"Z2RFRO1"	Q 38.0	BOOL	// [Z2ZB.M07]: SAFETY COMMON 1 (RESERVA)
"Z2RFRO2"	Q 38.1	BOOL	// [Z2ZB.M07]: SAFETY COMMON 2 (Z2ES)
"Z2ZB_M07_R1"	Q 38.2	BOOL	// [Z2ZB.M07]: RESERVA
"Z2EV7b"	Q 38.3	BOOL	// [Z2ZB.M07]: Z2 EV 7 bar
"Z3RFRO1"	Q 47.0	BOOL	// (Z2ZB.M09): RELE COMUN DE SEGURIDAD (Z3AU)
"Z3RFRO2"	Q 47.1	BOOL	// (Z2ZB.M09): RELE COMUN DE SEGURIDAD (Z3ES)
"Z3EV7B"	Q 47.3	BOOL	// (Z2ZB.M09): EV 7 BARS
"A0SB_M04_R1"	Q 70.0	BOOL	// [A0SB.M04]: RESERVA
"A0SB_M04_R2"	Q 70.1	BOOL	// [A0SB.M04]: RESERVA
"A0SB_M04_R3"	Q 70.2	BOOL	// [A0SB.M04]: RESERVA
"A0SB_M04_R4"	Q 70.3	BOOL	// [A0SB.M04]: RESERVA
"A0SB_M04_R5"	Q 70.4	BOOL	// [A0SB.M04]: RESERVA
"A0SB_M04_R6"	Q 70.5	BOOL	// [A0SB.M04]: RESERVA
"A0SB_M04_R7"	Q 70.6	BOOL	// [A0SB.M04]: RESERVA
"A0SB_M04_R8"	Q 70.7	BOOL	// [A0SB.M04]: RESERVA
"A0VAT"	Q 71.0	BOOL	// [A0SB.M06]: A0 WORK AUTHORIZATION LAMP 1 (GREEN)
"A0VIT"	Q 71.1	BOOL	// [A0SB.M06]: A0 WORK PROHIBITION LAMP 1 (RED)
"A0VDF"	Q 71.2	BOOL	// [A0SB.M06]: A0 DEFAULT LAMP 1 (ORANGE)
"A0SB_M06_R1"	Q 71.3	BOOL	// [A0SB.M06]: RESERVA
"A0SB_M06_R2"	Q 71.4	BOOL	// [A0SB.M06]: RESERVA
"A0SB_M06_R3"	Q 71.5	BOOL	// [A0SB.M06]: RESERVA
"A0SB_M06_R4"	Q 71.6	BOOL	// [A0SB.M06]: RESERVA
"A0SB_M06_R5"	Q 71.7	BOOL	// [A0SB.M06]: RESERVA
"A0RFRO1"	Q 90.0	BOOL	// [A0SB.M11]: A0 SAFETY COMMON 3 (FRO1)
"A0RFRO2"	Q 90.1	BOOL	// [A0SB.M11]: A0 SAFETY COMMON 4 (FRO2)
"A0RFRO3"	Q 90.2	BOOL	// [A0SB.M11]: A0 SAFETY COMMON 5 (FRO3)
"A0SB_M11_R1"	Q 90.3	BOOL	// [A0SB.M11]: RESERVA
"B0SB_M04_R1"	Q 110.0	BOOL	// [B0SB.M04]: RESERVA
"B0SB_M04_R2"	Q 110.1	BOOL	// [B0SB.M04]: RESERVA
"B0SB_M04_R3"	Q 110.2	BOOL	// [B0SB.M04]: RESERVA
"B0SB_M04_R4"	Q 110.3	BOOL	// [B0SB.M04]: RESERVA
"B0SB_M04_R5"	Q 110.4	BOOL	// [B0SB.M04]: RESERVA
"B0SB_M04_R6"	Q 110.5	BOOL	// [B0SB.M04]: RESERVA
"B0SB_M04_R7"	Q 110.6	BOOL	// [B0SB.M04]: RESERVA
"B0SB_M04_R8"	Q 110.7	BOOL	// [B0SB.M04]: RESERVA
"B0VAT"	Q 111.0	BOOL	// [B0SB.M06]: B0 WORK AUTHORIZATION LAMP 1 (GREEN)
"B0VIT"	Q 111.1	BOOL	// [B0SB.M06]: B0 WORK PROHIBITION LAMP 1 (RED)
"B0VDF"	Q 111.2	BOOL	// [B0SB.M06]: B0 DEFAULT LAMP 1 (ORANGE)
"B0SB_M06_R1"	Q 111.3	BOOL	// [B0SB.M06]: RESERVA
"B0SB_M06_R2"	Q 111.4	BOOL	// [B0SB.M06]: RESERVA
"B0SB_M06_R3"	Q 111.5	BOOL	// [B0SB.M06]: RESERVA
"B0SB_M06_R4"	Q 111.6	BOOL	// [B0SB.M06]: RESERVA
"B0SB_M06_R5"	Q 111.7	BOOL	// [B0SB.M06]: RESERVA
"B0SB_M11_R1"	Q 130.3	BOOL	// [B0SB.M11]: RESERVA
"C0SB_M04_R1"	Q 150.0	BOOL	// [C0SB.M04]: RESERVA
"C0SB_M04_R2"	Q 150.1	BOOL	// [C0SB.M04]: RESERVA
"C0SB_M04_R3"	Q 150.2	BOOL	// [C0SB.M04]: RESERVA
"C0SB_M04_R4"	Q 150.3	BOOL	// [C0SB.M04]: RESERVA
"C0SB_M04_R5"	Q 150.4	BOOL	// [C0SB.M04]: RESERVA
"C0SB_M04_R6"	Q 150.5	BOOL	// [C0SB.M04]: RESERVA
"C0SB_M04_R7"	Q 150.6	BOOL	// [C0SB.M04]: RESERVA
"C0SB_M04_R8"	Q 150.7	BOOL	// [C0SB.M04]: RESERVA
"C0VAT"	Q 151.0	BOOL	// [C0SB.M06]: C0 WORK AUTHORIZATION LAMP 1 (GREEN)
"C0VIT"	Q 151.1	BOOL	// [C0SB.M06]: C0 WORK PROHIBITION LAMP 1 (RED)
"C0VDF"	Q 151.2	BOOL	// [C0SB.M06]: C0 DEFAULT LAMP 1 (ORANGE)
"C0SB_M06_R1"	Q 151.3	BOOL	// [C0SB.M06]: RESERVA
"C0SB_M06_R2"	Q 151.4	BOOL	// [C0SB.M06]: RESERVA
"C0SB_M06_R3"	Q 151.5	BOOL	// [C0SB.M06]: RESERVA
"C0SB_M06_R4"	Q 151.6	BOOL	// [C0SB.M06]: RESERVA
"C0SB_M06_R5"	Q 151.7	BOOL	// [C0SB.M06]: RESERVA
"C0SB_M11_R1"	Q 170.3	BOOL	// [C0SB.M11]: RESERVA
"D0SB_M04_R1"	Q 190.0	BOOL	// [D0SB.M04]: RESERVA
"D0SB_M04_R2"	Q 190.1	BOOL	// [D0SB.M04]: RESERVA
"D0SB_M04_R3"	Q 190.2	BOOL	// [D0SB.M04]: RESERVA
"D0SB_M04_R4"	Q 190.3	BOOL	// [D0SB.M04]: RESERVA
"D0SB_M04_R5"	Q 190.4	BOOL	// [D0SB.M04]: RESERVA
"D0SB_M04_R6"	Q 190.5	BOOL	// [D0SB.M04]: RESERVA
"D0SB_M04_R7"	Q 190.6	BOOL	// [D0SB.M04]: RESERVA
"D0SB_M04_R8"	Q 190.7	BOOL	// [D0SB.M04]: RESERVA
"D0VAT"	Q 191.0	BOOL	// [D0SB.M06]: D0 WORK AUTHORIZATION LAMP 1 (GREEN)
"D0VIT"	Q 191.1	BOOL	// [D0SB.M06]: D0 WORK PROHIBITION LAMP 1 (RED)
"D0VDF"	Q 191.2	BOOL	// [D0SB.M06]: D0 DEFAULT LAMP 1 (ORANGE)
"D0LPDPY"	Q 191.3	BOOL	// [D0SB.M06]: LAMPADA DEFEITO POKAYOKE
"D0SRDPY"	Q 191.4	BOOL	// [D0SB.M06]: SIRENE DEFEITO POKAYOKE
"TR0VAT"	Q 191.5	BOOL	// [D0SB.M06]: TR0 LAMP(GREEN)
"TR0VIT"	Q 191.6	BOOL	// [D0SB.M06]: TR0 LAMP (RED)
"D0SB_M06_R5"	Q 191.7	BOOL	// [D0SB.M06]: RESERVA
"D0RFRO1"	Q 210.0	BOOL	// [D0SB.M11]: D0 SAFETY COMMON 3 (FRO1)
"D0RFRO2"	Q 210.1	BOOL	// [D0SB.M11]: D0 SAFETY COMMON 4 (FRO2)
"D0RFRO3"	Q 210.2	BOOL	// [D0SB.M11]: D0 SAFETY COMMON 5 (FRO3)
"D0SB_M11_R1"	Q 210.3	BOOL	// [D0SB.M11]: RESERVA
"E0SB_M04_R1"	Q 230.0	BOOL	// [E0SB.M04]: RESERVA
"E0SB_M04_R2"	Q 230.1	BOOL	// [E0SB.M04]: RESERVA
"E0SB_M04_R3"	Q 230.2	BOOL	// [E0SB.M04]: RESERVA
"E0SB_M04_R4"	Q 230.3	BOOL	// [E0SB.M04]: RESERVA
"E0SB_M04_R5"	Q 230.4	BOOL	// [E0SB.M04]: RESERVA
"E0SB_M04_R6"	Q 230.5	BOOL	// [E0SB.M04]: RESERVA
"E0SB_M04_R7"	Q 230.6	BOOL	// [E0SB.M04]: RESERVA
"E0SB_M04_R8"	Q 230.7	BOOL	// [E0SB.M04]: RESERVA
"E0VAT"	Q 231.0	BOOL	// [E0SB.M06]: E0 WORK AUTHORIZATION LAMP 1 (GREEN)
"E0VIT"	Q 231.1	BOOL	// [E0SB.M06]: E0 WORK PROHIBITION LAMP 1 (RED)
"E0VDF"	Q 231.2	BOOL	// [E0SB.M06]: E0 DEFAULT LAMP 1 (ORANGE)
"E0SB_M06_R1"	Q 231.3	BOOL	// [E0SB.M06]: RESERVA
"E0SB_M06_R2"	Q 231.4	BOOL	// [E0SB.M06]: RESERVA
"E0SB_M06_R3"	Q 231.5	BOOL	// [E0SB.M06]: RESERVA
"E0SB_M06_R4"	Q 231.6	BOOL	// [E0SB.M06]: RESERVA
"E0SB_M06_R5"	Q 231.7	BOOL	// [E0SB.M06]: RESERVA
"E0SB_M11_R1"	Q 250.3	BOOL	// [E0SB.M11]: RESERVA
"F0SB_M04_R1"	Q 270.0	BOOL	// [F0SB.M04]: RESERVA
"F0SB_M04_R2"	Q 270.1	BOOL	// [F0SB.M04]: RESERVA
"F0SB_M04_R3"	Q 270.2	BOOL	// [F0SB.M04]: RESERVA
"F0SB_M04_R4"	Q 270.3	BOOL	// [F0SB.M04]: RESERVA
"F0SB_M04_R5"	Q 270.4	BOOL	// [F0SB.M04]: RESERVA
"F0SB_M04_R6"	Q 270.5	BOOL	// [F0SB.M04]: RESERVA
"F0SB_M04_R7"	Q 270.6	BOOL	// [F0SB.M04]: RESERVA
"F0SB_M04_R8"	Q 270.7	BOOL	// [F0SB.M04]: RESERVA
"F0VAT"	Q 271.0	BOOL	// [F0SB.M06]: F0 WORK AUTHORIZATION LAMP 1 (GREEN)
"F0VIT"	Q 271.1	BOOL	// [F0SB.M06]: F0 WORK PROHIBITION LAMP 1 (RED)
"F0VDF"	Q 271.2	BOOL	// [F0SB.M06]: F0 DEFAULT LAMP 1 (ORANGE)
"F0SB_M06_R1"	Q 271.3	BOOL	// [F0SB.M06]: RESERVA
"F0SB_M06_R2"	Q 271.4	BOOL	// [F0SB.M06]: RESERVA
"F0SB_M06_R3"	Q 271.5	BOOL	// [F0SB.M06]: RESERVA
"F0SB_M06_R4"	Q 271.6	BOOL	// [F0SB.M06]: RESERVA
"F0SB_M06_R5"	Q 271.7	BOOL	// [F0SB.M06]: RESERVA
"F0RFRO1"	Q 290.0	BOOL	// [F0SB.M11]: F0 SAFETY COMMON 3 (F0SOP)
"F0RFRO2"	Q 290.1	BOOL	// [F0SB.M11]: F0 SAFETY COMMON 4 (F0)
"F0RFRO3"	Q 290.2	BOOL	// [F0SB.M11]: F0 SAFETY COMMON 5 (F0)
"F0SB_M11_R1"	Q 290.3	BOOL	// [F0SB.M11]: RESERVA
"G0SB_M04_R1"	Q 310.0	BOOL	// [G0SB.M04]: RESERVA
"G0SB_M04_R2"	Q 310.1	BOOL	// [G0SB.M04]: RESERVA
"G0SB_M04_R3"	Q 310.2	BOOL	// [G0SB.M04]: RESERVA
"G0SB_M04_R4"	Q 310.3	BOOL	// [G0SB.M04]: RESERVA
"G0SB_M04_R5"	Q 310.4	BOOL	// [G0SB.M04]: RESERVA
"G0SB_M04_R6"	Q 310.5	BOOL	// [G0SB.M04]: RESERVA
"G0SB_M04_R7"	Q 310.6	BOOL	// [G0SB.M04]: RESERVA
"G0SB_M04_R8"	Q 310.7	BOOL	// [G0SB.M04]: RESERVA
"G0VAT"	Q 311.0	BOOL	// [G0SB.M06]: G0 WORK AUTHORIZATION LAMP 1 (GREEN)
"G0VIT"	Q 311.1	BOOL	// [G0SB.M06]: G0 WORK PROHIBITION LAMP 1 (RED)
"G0VDF"	Q 311.2	BOOL	// [G0SB.M06]: G0 DEFAULT LAMP 1 (ORANGE)
"G0SB_M06_R1"	Q 311.3	BOOL	// [G0SB.M06]: RESERVA
"G0SB_M06_R2"	Q 311.4	BOOL	// [G0SB.M06]: RESERVA
"G0SB_M06_R3"	Q 311.5	BOOL	// [G0SB.M06]: RESERVA
"G0SB_M06_R4"	Q 311.6	BOOL	// [G0SB.M06]: RESERVA
"G0SB_M06_R5"	Q 311.7	BOOL	// [G0SB.M06]: RESERVA
"G0SB_M11_R1"	Q 330.3	BOOL	// [G0SB.M11]: RESERVA
"K0SB_M04_R1"	Q 380.0	BOOL	// [K0SB.M04]: RESERVA
"K0SB_M04_R2"	Q 380.1	BOOL	// [K0SB.M04]: RESERVA
"K0SB_M04_R3"	Q 380.2	BOOL	// [K0SB.M04]: RESERVA
"K0SB_M04_R4"	Q 380.3	BOOL	// [K0SB.M04]: RESERVA
"K0SB_M04_R5"	Q 380.4	BOOL	// [K0SB.M04]: RESERVA
"K0SB_M04_R6"	Q 380.5	BOOL	// [K0SB.M04]: RESERVA
"K0SB_M04_R7"	Q 380.6	BOOL	// [K0SB.M04]: RESERVA
"KOSB_M04_R8"	Q 380.7	BOOL	// [K0SB.M04]: RESERVA
"K0VAT"	Q 381.0	BOOL	// [K0SB.M06]: C0 WORK AUTHORIZATION LAMP 1 (GREEN)
"K0VIT"	Q 381.1	BOOL	// [K0SB.M06]: C0 WORK PROHIBITION LAMP 1 (RED)
"K0VDF"	Q 381.2	BOOL	// [K0SB.M06]: C0 DEFAULT LAMP 1 (ORANGE)
"K0SB_M06_R1"	Q 381.3	BOOL	// [K0SB.M06]: RESERVA
"K0SB_M06_R2"	Q 381.4	BOOL	// [K0SB.M06]: RESERVA
"K0SB_M06_R3"	Q 381.5	BOOL	// [K0SB.M06]: RESERVA
"K0SB_M06_R4"	Q 381.6	BOOL	// [K0SB.M06]: RESERVA
"K0SB_M06_R5"	Q 381.7	BOOL	// [K0SB.M06]: RESERVA
"K0RFRO1"	Q 400.0	BOOL	// [K0SB.M11]: K0 SAFETY COMMON 3 (K0SOP)
"K0RFRO2"	Q 400.1	BOOL	// [K0SB.M11]: K0 SAFETY COMMON 4 (K0SOP)
"K0RFRO3"	Q 400.2	BOOL	// [K0SB.M11]: K0 SAFETY COMMON 5 (K0SOP)
"K0SB_M11_R1"	Q 400.3	BOOL	// [K0SB.M11]: RESERVA
"A0EAPLA"	Q 500.0	BOOL	// [A0IM1.A0S11]: A0: EV AVANÇO PILOTO A
"A0EASRB"	Q 500.1	BOOL	// [A0IM1.A0S11]: A0: EV AVANÇO SERRAGE MANUAL B
"A0IM_A0S11_R1"	Q 500.2	BOOL	// [A0IM1.A0S11]: RESERVA
"A0EASRD"	Q 500.3	BOOL	// [A0IM1.A0S11]: A0: EV AVANÇO SERRAGE D
"A0ERPLA"	Q 500.4	BOOL	// [A0IM1.A0S11]: A0: EV RECUO PILOTO A
"A0ERSRB"	Q 500.5	BOOL	// [A0IM1.A0S11]: A0: EV RECUO SERRAGE MANUAL B
"A0IM_A0S11_R2"	Q 500.6	BOOL	// [A0IM1.A0S11]: RESERVA
"A0ERSRD"	Q 500.7	BOOL	// [A0IM1.A0S11]: A0: EV RECUO SERRAGE D
"A0EAPLE"	Q 501.0	BOOL	// [A0IM1.A0S12]: A0: EV AVANÇO PILOTO E
"A0IM_A0S12_R5"	Q 501.1	BOOL	// [A0IM1.A0S12]: RESERVA
"A0IM_A0S12_R3"	Q 501.2	BOOL	// [A0IM1.A0S12]: RESERVA
"A0IM_A0S12_R4"	Q 501.3	BOOL	// [A0IM1.A0S12]: RESERVA
"A0ERPLE"	Q 501.4	BOOL	// [A0IM1.A0S12]: A0: EV RECUO PILOTO E
"A0IM_A0S12_R6"	Q 501.5	BOOL	// [A0IM1.A0S12]: RESERVA
"A0IM_A0S12_R7"	Q 501.6	BOOL	// [A0IM1.A0S12]: RESERVA
"A0IM_A0S12_R8"	Q 501.7	BOOL	// [A0IM1.A0S12]: RESERVA
"B0EAPLA"	Q 520.0	BOOL	// [B0IM1.B0S11]: B0: EV AVANÇO PILOTO A
"B0EASRB"	Q 520.1	BOOL	// [B0IM1.B0S11]: B0: EV AVANÇO SERRAGE B
"B0IM_B0S11_R1"	Q 520.2	BOOL	// [B0IM1.B0S11]: RESERVA
"B0IM_B0S11_R2"	Q 520.3	BOOL	// [B0IM1.B0S11]: RESERVA
"B0ERPLA"	Q 520.4	BOOL	// [B0IM1.B0S11]: B0: EV RECUO PILOTO A
"B0ERSRB"	Q 520.5	BOOL	// [B0IM1.B0S11]: D0: EV RECUO SERRAGE B
"B0IM_B0S11_R3"	Q 520.6	BOOL	// [B0IM1.B0S11]: RESERVA
"B0IM_B0S11_R4"	Q 520.7	BOOL	// [B0IM1.B0S11]: RESERVA
"D0EAPLA"	Q 560.0	BOOL	// [D0IM1.D0S11]: D0: EV AVANÇO PILOTO A
"D0EACAB"	Q 560.1	BOOL	// [D0IM1.D0S11]: D0:EV AVANÇO CARRO B
"D0EASRC"	Q 560.2	BOOL	// [D0IM1.D0S11]: D0: EV AVANÇO SERRAGE C
"D0EASRD"	Q 560.3	BOOL	// [D0IM1.D0S11]: D0: EV AVANÇO SERRAGE D
"D0ERPLA"	Q 560.4	BOOL	// [D0IM1.D0S11]: D0: EV RECUO PILOTO A
"D0ERCAB"	Q 560.5	BOOL	// [D0IM1.D0S11]: D0:EV RECUO CARRO B
"D0ERSRC"	Q 560.6	BOOL	// [D0IM1.D0S11]: D0: EV RECUO SERRAGE C
"D0ERSRD"	Q 560.7	BOOL	// [D0IM1.D0S11]: D0: EV RECUO SERRAGE D
"D0EACAB1"	Q 561.0	BOOL	// [D0IM1.D0S12]: D0:EV FREIO D0CAB1
"D0EAPLE"	Q 561.1	BOOL	// [D0IM1.D0S12]: D0: EV AVANÇO PILOTO E
"D0EASRMF"	Q 561.2	BOOL	// [D0IM1.D0S12]:  ElectroValvula Avance SRM1
"D0IM_D0S12_R4"	Q 561.3	BOOL	// [D0IM1.D0S12]: RESERVA
"D0ERCAB1"	Q 561.4	BOOL	// [D0IM1.D0S12]: D0:EV RECUO CARRO B1 (FREIO)
"D0ERPLE"	Q 561.5	BOOL	// [D0IM1.D0S12]: D0: EV RECUO PILOTO E
"D0ERSRMF"	Q 561.6	BOOL	// [D0IM1.D0S12]: [D0IM1.D0S12]:  ElectroValvula Retroceso SRM1
"D0IM_D0S12_R8"	Q 561.7	BOOL	// [D0IM1.D0S12]: RESERVA
"E0EAPLA"	Q 580.0	BOOL	// [E0IM1.E0S11]: E0: EV AVANÇO PILOTO A
"E0EASRB"	Q 580.1	BOOL	// [E0IM1.E0S11]: E0: EV AVANÇO SERRAGE B
"E0IM_E0S11_R1"	Q 580.2	BOOL	// [E0IM1.E0S11]: RESERVA
"E0IM_E0S11_R2"	Q 580.3	BOOL	// [E0IM1.E0S11]: RESERVA
"E0ERPLA"	Q 580.4	BOOL	// [E0IM1.E0S11]: E0: EV RECUO PILOTO A
"E0ERSRB"	Q 580.5	BOOL	// [E0IM1.E0S11]: E0: EV RECUO SERRAGE B
"E0IM_E0S11_R3"	Q 580.6	BOOL	// [E0IM1.E0S11]: RESERVA
"E0IM_E0S11_R4"	Q 580.7	BOOL	// [E0IM1.E0S11]: RESERVA
"F0EAPLA"	Q 600.0	BOOL	// [F0IM1.F0S11]: F0: EV AVANÇO PILOTO A
"F0EASRB"	Q 600.1	BOOL	// [F0IM1.F0S11]: F0: EV AVANÇO SERRAGE MANUAL B
"F0ERSRMB"	Q 600.2	BOOL	// [F0IM1.F0S11]: F0: EV RECUO SERRAGE MANUAL B
"F0EASRD"	Q 600.3	BOOL	// [F0IM1.F0S11]: F0: EV AVANÇO SERRAGE D
"F0ERPLA"	Q 600.4	BOOL	// [F0IM1.F0S11]: F0: EV RECUO PILOTO A
"F0ERSRB"	Q 600.5	BOOL	// [F0IM1.F0S11]: F0: EV RECUO SERRAGE B
"F0IM_F0S11_R1"	Q 600.6	BOOL	// [F0IM1.F0S11]: RESERVA
"F0ERSRD"	Q 600.7	BOOL	// [F0IM1.F0S11]: F0: EV RECUO SERRAGE D
"F0ERRCE"	Q 601.0	BOOL	// [F0IM1.F0S12]: F0: EV RECUO RETACAGE E
"F0EACAF"	Q 601.1	BOOL	// [F0IM1.F0S12]: F0: EV AVANÇO CARRO F
"F0EARCF1"	Q 601.2	BOOL	// [F0IM1.F0S12]: F0: EV AVANÇO RETACAGE F1
"F0IM_F0S12_R1"	Q 601.3	BOOL	// [F0IM1.F0S12]: RESERVA
"F0EARCE"	Q 601.4	BOOL	// [F0IM1.F0S12]: F0: EV AVANÇO RETACAGE E
"F0ERCAF"	Q 601.5	BOOL	// [F0IM1.F0S12]: F0: EV RECUO CARRO F
"F0IM_F0S12_R2"	Q 601.6	BOOL	// [F0IM1.F0S12]: RESERVA
"F0IM_F0S12_R3"	Q 601.7	BOOL	// [F0IM1.F0S12]: RESERVA
"G0EAPLA"	Q 620.0	BOOL	// [G0IM1.G0S11]: G0: EV AVANÇO PILOTO A
"G0EASRB"	Q 620.1	BOOL	// [G0IM1.G0S11]: G0: EV AVANÇO SERRAGE B
"G0IM_G0S13_R1"	Q 620.2	BOOL	// [G0IM1.G0S11]: RESERVA
"G0IM_G0S13_R2"	Q 620.3	BOOL	// [G0IM1.G0S11]: RESERVA
"G0ERPLA"	Q 620.4	BOOL	// [G0IM1.G0S11]: G0: EV RECUO PILOTO A
"G0ERSRB"	Q 620.5	BOOL	// [G0IM1.G0S11]: G0: EV RECUO SERRAGE B
"G0IM_G0S13_R3"	Q 620.6	BOOL	// [G0IM1.G0S11]: RESERVA
"G0IM_G0S13_R4"	Q 620.7	BOOL	// [G0IM1.G0S11]: RESERVA
"RESERVA-"	Q 640.7	BOOL	// [H0IM1.H0S11]: H0: RESERVA
"K0EASR1"	Q 650.0	BOOL	// [K0TDS1] K0: EV AVANCE SR1
"K0ERSR1"	Q 650.1	BOOL	// [K0TDS1] K0: EV RETROCESO SR1
"K0EASR2"	Q 650.2	BOOL	// [K0TDS1] K0: EV AVANCE SR2
"K0ERSR2"	Q 650.3	BOOL	// [K0TDS1] K0: EV RETROCESO SR2
"K0S11_RESERVA1"	Q 650.4	BOOL
"K0S11_RESERVA2"	Q 650.5	BOOL
"K0EASR3"	Q 650.6	BOOL	// [K0TDS1] K0: EV AVANCE SR3
"K0ERSR3"	Q 650.7	BOOL	// [K0TDS1] K0: EV RETROCESO SR3
"K0_VVAL"	Q 656.0	BOOL	// [K0A2] Habilitacion de 24V Valvulas CPX K0TDS1
"K0EVCPX"	Q 656.1	BOOL	// [K0A2] ELECTROVÁLVULA CPX K0TDS1
"Z2RCM"	Q 800.7	BOOL	// [Z2ZB.M05]: Z2 GROUND CONTROL RELAY
"Z2RSC1"	Q 815.0	BOOL	// [Z2ZB.M09]: RELAY SAFETY COMMON 1 (AU)
"Z2RES"	Q 815.1	BOOL	// [Z2ZB.M09]: RELAY SAFETY COMMON 2 (ES)
"Z2RFZ"	Q 815.2	BOOL	// [Z2ZB.M09]: RELAY SAFETY COMMON 3 (RFZ)
"Z2RSC4"	Q 815.3	BOOL	// [Z2ZB.M09]: RELAY SAFETY COMMON 4 (SC4)
"B1OP1VAT"	Q 821.0	BOOL	// B1 Lampara autorizacion de trabajo
"B1OP1VIT"	Q 821.1	BOOL	// B1 Lampara de prohibicion de trabajo
"B1OP1VDF"	Q 821.2	BOOL	// B1 Lampara de defecto
"B0RFRO1"	Q 841.0	BOOL	// [B0SB.M11]: B0 SAFETY COMMON 3 (FRO1)
"B0RFRO2"	Q 841.1	BOOL	// [B0SB.M11]: B0 SAFETY COMMON 4 (FRO2)
"B0RFRO3"	Q 841.2	BOOL	// [B0SB.M11]: B0 SAFETY COMMON 5 (FRO3)
"C1OP1VAT"	Q 851.0	BOOL	// C1 Lampara autorizacion de trabajo
"C1OP1VIT"	Q 851.1	BOOL	// C1 Lampara de prohibicion de trabajo
"C1OP1VDF"	Q 851.2	BOOL	// C1 Lampara de defecto
"C0RFRO1"	Q 871.0	BOOL	// [C0SB.M11]: C0 SAFETY COMMON 3 (C0SOP)
"C0RFRO2"	Q 871.1	BOOL	// [C0SB.M11]: C0 SAFETY COMMON 4 (C0)
"C0RFRO3"	Q 871.2	BOOL	// [C0SB.M11]: C0 SAFETY COMMON 5 (C0)
"E1OP1VAT"	Q 881.0	BOOL	// E1 Lampara autorizacion de trabajo
"E1OP1VIT"	Q 881.1	BOOL	// E1 Lampara de prohibicion de trabajo
"E1OP1VDF"	Q 881.2	BOOL	// E1 Lampara de defecto
"E2OP2VAT"	Q 881.5	BOOL
"E2OP2VIT"	Q 881.6	BOOL
"E0RFRO1"	Q 901.0	BOOL	// [E0SB.M11]: E0 SAFETY COMMON 3 ( E0SOP)
"E0RFRO2"	Q 901.1	BOOL	// [E0SB.M11]: E0 SAFETY COMMON 4 ( E0)
"E0RFRO3"	Q 901.2	BOOL	// [E0SB.M11]: E0 SAFETY COMMON 5 ( E0)
"G1OP1VAT"	Q 911.0	BOOL	// B1 Lampara autorizacion de trabajo
"G1OP1VIT"	Q 911.1	BOOL	// B1 Lampara de prohibicion de trabajo
"G1OP1VDF"	Q 911.2	BOOL	// B1 Lampara de defecto
"G0RFRO1"	Q 931.0	BOOL	// [G0SB.M11]: G0 SAFETY COMMON 3 (G0SOP)
"G0RFRO2"	Q 931.1	BOOL	// [G0SB.M11]: G0 SAFETY COMMON 4 (G0)
"G0RFRO3"	Q 931.2	BOOL	// [G0SB.M11]: G0 SAFETY COMMON 5 (G0)
"J1OP1VAT"	Q 940.0	BOOL	// J1 Lampara autorizacion de trabajo
"J1OP1VIT"	Q 940.1	BOOL	// J1 Lampara de prohibicion de trabajo
"J1OP1VDF"	Q 940.2	BOOL	// J1 Lampara de defecto
"B0EAPL1"	Q 950.0	BOOL	// [B0DTS1]: B0: EV AVANCE PL1
"B0ERPL1"	Q 950.1	BOOL	// [B0DTS1]: B0: EV RETROCESO PL1
"B0EASR2"	Q 950.2	BOOL	// [B0DTS1]: B0: EV AVANCE SR2
"B0ERSR2"	Q 950.3	BOOL	// [B0DTS1]: B0: EV RETROCESO SR2
"B0EASR3"	Q 950.4	BOOL	// [B0DTS1]: B0: EV AVANCE SR3
"B0ERSR3"	Q 950.5	BOOL	// [B0DTS1]: B0: EV RETROCESO SR3
"C0EAPL1"	Q 960.0	BOOL	// [C0DTS1]: C0: EV AVANCE PL1
"C0ERPL1"	Q 960.1	BOOL	// [C0DTS1]: C0: EV RETROCESO PL1
"C0EASR2"	Q 961.2	BOOL	// [C0DTS1]: C0: EV AVANCE SR2
"C0ERSR2"	Q 961.3	BOOL	// [C0DTS1]: C0: EV RETROCESO SR2
"C0EASR3"	Q 961.4	BOOL	// [C0DTS1]: C0: EV AVANCE SR3
"C0ERSR3"	Q 961.5	BOOL	// [C0DTS1]: C0: EV RETROCESO SR3
"E0EASR1"	Q 1040.0	BOOL	// [E0TDS1]: E0: EV AVANCE SR1
"E0ERSR1"	Q 1040.1	BOOL	// [E0TDS1]: E0: EV RETROCESO SR1
"E0EASR2"	Q 1040.2	BOOL	// [E0TDS1]: E0: EV AVANCE SR2
"E0ERSR2"	Q 1040.3	BOOL	// [E0TDS1]: E0: EV RETROCESO SR2
"E0EASR3"	Q 1040.4	BOOL	// [E0TDS1]: E0: EV AVANCE SR3
"E0ERSR3"	Q 1040.5	BOOL	// [E0TDS1]: E0: EV RETROCESO SR3
"E0EAVU4"	Q 1040.6	BOOL	// [E0TDS1]: E0: EV AVANCE VU4
"E0ERVU4"	Q 1040.7	BOOL	// [E0TDS1]: E0: EV RETROCESO VU4
"E0EAVU5"	Q 1041.0	BOOL	// [E0TDS1]: E0: EV AVANCE VU5
"E0ERVU5"	Q 1041.1	BOOL	// [E0TDS1]: E0: EV RETROCESO VU5
"E0EASR6"	Q 1041.2	BOOL	// [E0TDS1]: E0: EV AVANCE SR6
"E0ERSR6"	Q 1041.3	BOOL	// [E0TDS1]: E0: EV RETROCESO SR6
"G0EASR1"	Q 1060.0	BOOL	// [G0TDS1]: G0: EV AVANCE SR1
"G0ERSR1"	Q 1060.1	BOOL	// [G0TDS1]: G0: EV RETROCESO SR1
"G0EASR2"	Q 1060.2	BOOL	// [G0TDS1]: G0: EV AVANCE SR2
"G0ERSR2"	Q 1060.3	BOOL	// [G0TDS1]: G0: EV RETROCESO SR2
"G0EASR3"	Q 1060.4	BOOL	// [G0TDS1]: G0: EV AVANCE SR3
"G0ERSR3"	Q 1060.5	BOOL	// [G0TDS1]: G0: EV RETROCESO SR3
"L1VROC"	Q 1070.0	BOOL	// L1: LED BOTON RETORNO A ORIGEN
"L1VIT"	Q 1070.2	BOOL	// L1: LAMPARA DE PROHIBICION DE TRABAJO
"L1VDF"	Q 1070.3	BOOL	// L1: LAMPARA DE DEFECTO
"L1VAT"	Q 1070.4	BOOL	// L1: LAMPARA DE PROHIBICION DE TRABAJO
"L0EAPS1"	Q 1071.0	BOOL	// L0: Electrovalvula de avance PIN SHIFT 1
"L0ERPS1"	Q 1071.1	BOOL	// L0: Electrovalvula de retroceso PIN SHIFT 1
"L0EASR1"	Q 1071.2	BOOL	// L0: Electrovalvula de avance CLAMP 1
"L0ERSR1"	Q 1071.3	BOOL	// L0: Electrovalvula de retroceso CLAMP 1
"L0EASR2"	Q 1071.4	BOOL	// L0: Electrovalvula de avance CLAMP 2
"L0ERSR2"	Q 1071.5	BOOL	// L0: Electrovalvula de retroceso CLAMP 2
"L0EASR3"	Q 1071.6	BOOL	// L0: Electrovalvula de avance CLAMP 3
"L0ERSR3"	Q 1071.7	BOOL	// L0: Electrovalvula de retroceso CLAMP 3
"L0EAVU1"	Q 1072.0	BOOL	// L0: Electrovalvula de avance EJECTOR 1
"L0ERVU1"	Q 1072.1	BOOL	// L0: Electrovalvula de retroceso EJECTOR 1
"L0EAVU2"	Q 1072.2	BOOL	// L0: Electrovalvula de avance PINGYI 1
"L0ERVU2"	Q 1072.3	BOOL	// L0: Electrovalvula de retroceso PINGYI 1
"L0EASR4"	Q 1072.4	BOOL	// L0: ELECTROVALVULA DE AVANCE MOV SR4 (DETECTOR DPP15)
"L0ERSR4"	Q 1072.5	BOOL	// L0: ELECTROVALVULA DE AVANCE MOV SR4 (DETECTOR DPP15)
"FDIS_90_8_AckCan"	Q 1080.0	BOOL	// FESTO DI-Safe error de canal 90 - 8 L0
"FDIS_90_8_Pass"	Q 1080.1	BOOL	// FESTO DI-Safe 90 - 8 1 PASSIVATION PAR CANAL / 0 - PASSIVATION PAR MODULE
"L0SOP"	Q 1087.0	BOOL
"L024SV"	Q 1087.1	BOOL	// L0 24V SUPPLY FOR SOFSTART VALVE
"M1VROC"	Q 1100.0	BOOL	// M1: LAMPARA DE RETORNO AL ORIGEN
"M1VIT"	Q 1100.2	BOOL	// M1: LAMPARA DE PROHIBICION DE TRABAJO
"M1VDF"	Q 1100.3	BOOL	// M1: LAMPARA DE DEFECTO
"M1VAT"	Q 1100.4	BOOL	// M1: LAMPARA DE PERMISO DE TRABAJO
"FDIS_100_5_AckCan"	Q 1104.0	BOOL	// FESTO DI-Safe ERROR DE CANAL M0
"FDIS_100_5_Pass"	Q 1104.1	BOOL	// FESTO DI-Safe 1 - passivation par canal / 0 - passivation par module
"M0SOP"	Q 1111.0	BOOL
"M024SV"	Q 1111.1	BOOL	// M0 24V SUPPLY FOR SOFSTART VALVE
"M0EASR1"	Q 1117.0	BOOL	// M0: Electrovalvula avance HAND CLAMP 1
"M0ERSR1"	Q 1117.1	BOOL	// M0: Electrovalvula retroceso HAND CLAMP 1
"M0EASR2"	Q 1117.2	BOOL	// M0: Electrovalvula avance CLAMP 1
"M0ERSR2"	Q 1117.3	BOOL	// M0: Electrovalvula retroceso CLAMP 1
"M0EAVU1"	Q 1117.4	BOOL	// M0: Electrovalvula avance EJECTOR 1
"M0ERVU1"	Q 1117.5	BOOL	// M0: Electrovalvula retroceso EJECTOR 1
"N0EAPLC"	Q 1150.4	BOOL
"N0ERPLC"	Q 1150.5	BOOL
"N0EASRD"	Q 1150.6	BOOL
"N0ERSRD"	Q 1150.7	BOOL
"N0EASRE"	Q 1151.0	BOOL
"N0ERSRE"	Q 1151.1	BOOL
"N0EASRF"	Q 1151.2	BOOL
"N0ERSRF"	Q 1151.3	BOOL
"N0EACLH"	Q 1151.6	BOOL
"N0ERCLH"	Q 1151.7	BOOL
"N0EASRJ"	Q 1152.0	BOOL
"N0ERSRJ"	Q 1152.1	BOOL
"N0EACLK"	Q 1152.2	BOOL
"N0ERCLK"	Q 1152.3	BOOL
"N0EBLK"	Q 1152.4	BOOL	// ElectroValvula Bloqueti Cilindro K
"N1VDF"	Q 1155.0	BOOL	// N1: LAMPARA DE DEFECTO
"N1VAT"	Q 1155.1	BOOL	// N1: LAMPARA DE PERMISO DE TRABAJO
"N1VIT"	Q 1155.3	BOOL	// N1: LAMPARA DE PROHIBICION DE TRABAJO
"N0EAPLA"	Q 1156.0	BOOL
"N0ERPLA"	Q 1156.1	BOOL
"N0EACLB"	Q 1156.2	BOOL
"N0ERCLB"	Q 1156.3	BOOL
"N0EACLG"	Q 1156.4	BOOL
"N0ERCLG"	Q 1156.5	BOOL
"FDIS_110_5_AckCan"	Q 1158.0	BOOL	// FESTO DI-Safe ERROR DE CANAL M0
"FDIS_110_5_Pass"	Q 1158.1	BOOL	// FESTO DI-Safe 1 - passivation par canal / 0 - passivation par modul
"N0SOP"	Q 1165.0	BOOL	// N0IM1: COMUN SEGURIDAD OPERADO
"N0EVAIR"	Q 1165.1	BOOL	// N0 ELECTROVALVULA DE AIRE GENERAL
"FDIS_90_8_M"	QW 1081	INT	// FESTO DI-Safe 90-8 MODE L0
"FDIS_100_5_M"	QW 1105	INT	// FESTO DI-Safe 100 - 5 MODE
"FDIS_110_5_M"	QW 1159	INT	// FESTO DI-Safe 110 - 5 MODE
"TP"	SFB 3	SFB 3	// GENERATE A PULSE
"TON"	SFB 4	SFB 4	// GENERATE AN ON DELAY
"TOF"	SFB 5	SFB 5	// GENERATE AN OFF DELAY
"RDREC"	SFB 52	SFB 52	// READ A PROCESS DATA RECORD
"WRREC"	SFB 53	SFB 53	// WRITE A PROCESS DATA RECORD
"RALRM"	SFB 54	SFB 54	// Receive Alarm Data
"SET_CLK"	SFC 0	SFC 0	// SET SYSTEM CLOCK
"READ_CLK"	SFC 1	SFC 1	// READ SYSTEM CLOCK
"RD_SINFO"	SFC 6	SFC 6	// READ OB START INFORMATION
"D_ACT_DP"	SFC 12	SFC 12	// DEACTIVATING AND ACTIVATING DP SLAVES
"DPRD_DAT"	SFC 14	SFC 14	// READ CONSISTENT DATA OF A STANDARD DP SLAVE
"DPWR_DAT"	SFC 15	SFC 15	// WRITE CONSISTENT DATA TO A STANDARD DP SLAVE
"BLKMOV"	SFC 20	SFC 20	// COPY VARIABLES
"FILL"	SFC 21	SFC 21	// INITIALIZE A MEMORY AREA
"TEST_DB"	SFC 24	SFC 24	// TEST DATA BLOCK
"DIS_AIRT"	SFC 41	SFC 41	// DELAY THE HIGHER PRIORITY INTERRUPTS AND ASYNCHRONOUS ERRORS
"EN_AIRT"	SFC 42	SFC 42	// ENABLE HIGHER PRIORITY INTERRUPTS AND ASYNCHRONOUS ERRORS
"STP"	SFC 46	SFC 46	// CHANGE THE CPU TO STOP
"RDSYSST"	SFC 51	SFC 51	// READ A SYSTEM STATUS LIST OR PARTIAL LIST
"WR_REC"	SFC 58	SFC 58	// WRITE DATA RECORD
"RD_REC"	SFC 59	SFC 59	// READ A DATA RECORD
"TIME_TCK"	SFC 64	SFC 64	// READ THE SYSTEM TIME
"GEO_LOG"	SFC 70	SFC 70	// DETERMINE LOGICAL ADDRESS
"READ_DBL"	SFC 83	SFC 83	// READ DATA BLOCK OUT OF LOAD MEMORY
"WRIT_DBL"	SFC 84	SFC 84	// WRITE DATA BLOCK IN LOAD MEMORY
"DEL_SI"	SFC 106	SFC 106	// Deleting Dynamically Assigned System Instances
"ALARM_DQ"	SFC 107	SFC 107	// Creating Acknowledgeable Block-related Message
"ALARM_D"	SFC 108	SFC 108	// Creating Acknowledged Block-related Message
"LIEN_SEC"	UDT 1507	UDT 1507	// TABLE COMMUNE AUX BF_ZONE_PORTE1, BF_ZONE_RSEC1, BF_ZONE_MODE_IHM, BF_ZONE_AIR
"MOT_FONC_DPL"	UDT 1866	UDT 1866
"LIEN_PUP"	UDT 1988	UDT 1988	// Gestion des Modes et des pupitres de cde manu de la  zone (BF_ZONE_MODE_IHM)
"LIEN_ILOT"	UDT 2004	UDT 2004	// INFO CONTROL LINKED TO THE FACILITY (BF_ILOT)
"MOT_FONC_MP"	UDT 2041	UDT 2041	// INFO CONTROL OF A MOVEMENT (BF_MOUVMP1)
"MOT_FONC"	UDT 2042	UDT 2042	// INFO D'UN MOUVEMENT (BF_MOUV2P1,BF_MVSE2P1, BF_RB_COD_PREH_API)
"VAT_SIPTOL"	VAT 1	
"VAT_TALOA0"	VAT 2	
"VAT_BASE DE DADOS"	VAT 3	
"Z1T_TEMPOS"	VAT 4	
"Z2T_TEMPOS"	VAT 5	
"VAT_6"	VAT 6	
"acompanhamento zona 8"	VAT 7		// teste tucker
"TOMAS"	VAT 8	
"W0"	VAT 9	
"VAT_Z1_BOT_EMER"	VAT 10	
"VAT_Z2_BOT_EMER"	VAT 11		// BOTAO_DE_EMERGENCIA
"VAT_Z1_VALIDAÇÃO"	VAT 12	
"VAT_CDIV_2"	VAT 13	
"VAT_Z2_VALIDAÇÃO"	VAT 14	
"ELEV_CARREGAMENTO"	VAT 15	
"ELEV_DESCARREGAMENTO"	VAT 16	
"VAT_17"	VAT 17	
"TESTE_MODO_DEGR"	VAT 18	
"Z2_SIPTOL"	VAT 19	
"mostrar IIT"	VAT 20	
"tab_iit_2"	VAT 21	
"VAT_22"	VAT 22	
"afficher"	VAT 23	
"VAT_24"	VAT 24	
"SIPTOL_X52_X67_X60"	VAT 25	
"Z3_SIPTOL"	VAT 26		// VAT SIPTOL ZONA 3
"VAT_IIT"	VAT 27	
"VAT_Z1T"	VAT 28	
"SMP"	VAT 29	
"def_qbad"	VAT 30	
END_SYMBOL_TABLE
